// LS Electric XG5000 project: 과년69_3_A
// PLC NewPLC
// module base 0 slot 0: 입출력 모듈:XBC-DR20S (DC 24V 입력 12점, 릴레이 출력 8점)

PROGRAM NewProgram (task: 스캔 프로그램)

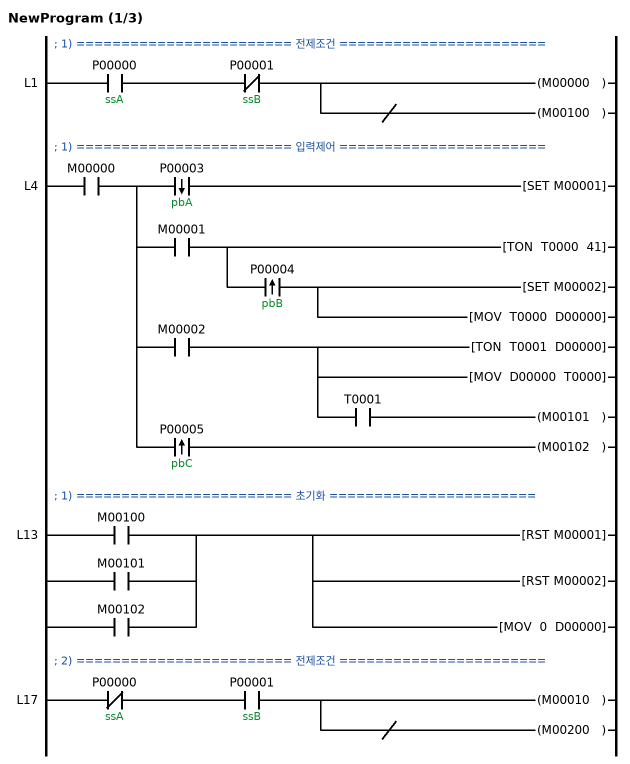
// 1) ======================== 전제조건 =======================
; L1
LOAD      P00000	// ssA
AND NOT   P00001	// ssB
OUT       M00000
NOT
OUT       M00100
// 1) ======================== 입력제어 =======================
; L4
LOAD      M00000
MPUSH
ANDN      P00003	// pbA
SET       M00001
MLOAD
AND       M00001
TON       T0000 41
ANDP      P00004	// pbB
SET       M00002
MOV       T0000 D00000
MLOAD
AND       M00002
TON       T0001 D00000
MOV       D00000 T0000
AND       T0001
OUT       M00101
MPOP
ANDP      P00005	// pbC
OUT       M00102
// 1) ======================== 초기화 =======================
; L13
LOAD      M00100
OR        M00101
OR        M00102
RST       M00001
RST       M00002
MOV       0 D00000
// 2) ======================== 전제조건 =======================
; L17
LOAD NOT  P00000	// ssA
AND       P00001	// ssB
OUT       M00010
NOT
OUT       M00200

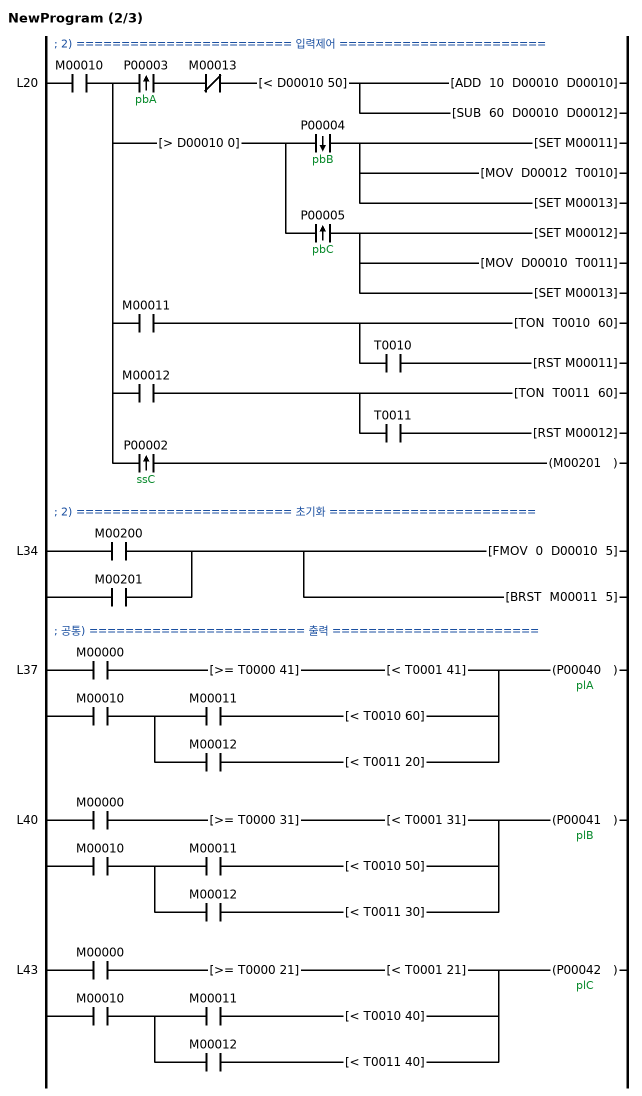
// 2) ======================== 입력제어 =======================
; L20
LOAD      M00010
MPUSH
ANDP      P00003	// pbA
AND NOT   M00013
AND<      D00010 50
ADD       10 D00010 D00010
SUB       60 D00010 D00012
MLOAD
AND>      D00010 0
MPUSH
ANDN      P00004	// pbB
SET       M00011
MOV       D00012 T0010
SET       M00013
MPOP
ANDP      P00005	// pbC
SET       M00012
MOV       D00010 T0011
SET       M00013
MLOAD
AND       M00011
TON       T0010 60
AND       T0010
RST       M00011
MLOAD
AND       M00012
TON       T0011 60
AND       T0011
RST       M00012
MPOP
ANDP      P00002	// ssC
OUT       M00201
// 2) ======================== 초기화 =======================
; L34
LOAD      M00200
OR        M00201
FMOV      0 D00010 5
BRST      M00011 5
// 공통) ======================== 출력 =======================
; L37
LOAD      M00000
AND>=     T0000 41
AND<      T0001 41
LOAD      M00010
LOAD      M00011
AND<      T0010 60
LOAD      M00012
AND<      T0011 20
OR LOAD
AND LOAD
OR LOAD
OUT       P00040	// plA
; L40
LOAD      M00000
AND>=     T0000 31
AND<      T0001 31
LOAD      M00010
LOAD      M00011
AND<      T0010 50
LOAD      M00012
AND<      T0011 30
OR LOAD
AND LOAD
OR LOAD
OUT       P00041	// plB
; L43
LOAD      M00000
AND>=     T0000 21
AND<      T0001 21
LOAD      M00010
LOAD      M00011
AND<      T0010 40
LOAD      M00012
AND<      T0011 40
OR LOAD
AND LOAD
OR LOAD
OUT       P00042	// plC

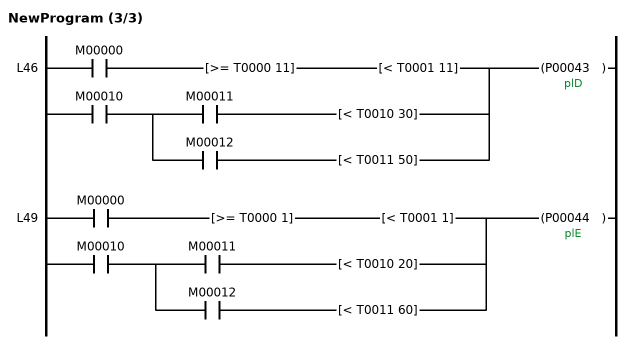
; L46
LOAD      M00000
AND>=     T0000 11
AND<      T0001 11
LOAD      M00010
LOAD      M00011
AND<      T0010 30
LOAD      M00012
AND<      T0011 50
OR LOAD
AND LOAD
OR LOAD
OUT       P00043	// plD
; L49
LOAD      M00000
AND>=     T0000 1
AND<      T0001 1
LOAD      M00010
LOAD      M00011
AND<      T0010 20
LOAD      M00012
AND<      T0011 60
OR LOAD
AND LOAD
OR LOAD
OUT       P00044	// plE